{attribute 'linkalways'} 
{attribute 'no_explicit_call' := 'This FB is a CLASS and must be accessed using methods or properties'}
{attribute 'enable_dynamic_creation'}
FUNCTION_BLOCK ChunkedResponsesMiddleware EXTENDS Middleware
VAR
	chunkedResponseManager : I_ChunkedResponseManager;
	config : I_ChunkedResponsesMiddlewareConfig;
END_VAR

METHOD FB_init : BOOL
VAR_INPUT
	bInitRetains : BOOL; // if TRUE, the retain variables are initialized (warm start / cold start)
	bInCopyCode : BOOL;  // if TRUE, the instance afterwards gets moved into the copy code (online change)
	ChunkedResponseManager : I_ChunkedResponseManager;
	Config : I_ChunkedResponsesMiddlewareConfig;
END_VAR
THIS^.chunkedResponseManager := ChunkedResponseManager;
THIS^.config := Config;
END_METHOD

METHOD PUBLIC Handle
VAR_INPUT
	Request : I_Request;
	Response : I_ServerResponse;
END_VAR
VAR
	chunkableServerResponse : ChunkableServerResponse(Response, chunkedResponseManager);
END_VAR
IF chunkedResponseManager.TryHandleIncomingRequest(Request, Response) THEN
	RETURN;
END_IF

Next(Request, chunkableServerResponse);
END_METHOD

METHOD PUBLIC UpdateConfig
VAR_INPUT
	Config : I_ChunkedResponsesMiddlewareConfig;
END_VAR
this^.config := Config;
END_METHOD

END_FUNCTION_BLOCK

(* stored: Version 1.1.0.1, ProductVersion 3.1.4024.12
   POU ChunkedResponsesMiddleware: Id {b4a4ecdd-bc41-4a65-a285-564fd7ee40d5}, SpecialFunc None
   Folder Constructor: Id {891d9d47-30b9-44e7-8b39-865cb2c8fb3e}
   Method FB_init: Id {057b0524-c39c-4f2e-9338-77dff1aeb7e9}
   Method Handle: Id {233b0b80-15cd-432e-b8d7-1d7e76c75590}
   Method UpdateConfig: Id {51266403-a36a-451e-bac8-aa23236cb9bb} *)
